// TIA Portal V19 export
FUNCTION "STOP PRODUCTION" : Void   // FC46, STL
TITLE = STOP PRODUCTION ASEPTIC TANK
{ S7_Optimized_Access := 'TRUE' }
NAME : SPROTNK
VERSION : 0.0
// Comment
// stored: AutoNumber false
BEGIN

NETWORK
TITLE = STOP PRODUCTION ASEPTIC TANK
// "M_PACK1", "M_PACK2", "M_PACK3", "M_PACK4" have been commented out to free up 
// outputs which were not wired, to be used for the Combi 512 Filler cip interface
      AN    "S0 STOP PRODUCTION TANK";
      R     "S1 STOP PRODUCTION TANK";
      R     "S2 STOP PRODUCTION TANK";
      BEC;
      A     "S1 STOP PRODUCTION TANK";
      JC    M001;
      R     "TANK STERILE";
      R     "MY0113";
      R     "MY0112";
      S     "MY0114";
      R     "MY0148";
      R     "IF_Device".V_09_30.IO.V._IO.IN.Activate;
      R     "IF_Device".V_09_31.IO.V._IO.IN.Activate;
      R     "TEST BARRIERS";
      R     "TEST FILLING PRESSURE";
//     R     "MM01.30"
      R     "START FILLING TANK";
      R     "STOP FILLING TANK";
      R     "MY0147";
      R     "M_AHV_READY";
//     R     "M_PACK1"
//     R     "M_PACK2"
//     R     "M_PACK3"
//     R     "M_PACK4"
      R     "DUMMY PROD. AT FILLING";
      R     "AGITATOR AUTOMATIC";
      R     "AGITATOR MANUEL";

//      A     "B01.66"
//      S     "A13-DRAIN THE TANK"
//      SET

      S     "S1 STOP PRODUCTION TANK";
      BEU;
M001: NOP   0;

NETWORK
TITLE = 
// Comment
      A     "S2 STOP PRODUCTION TANK";
      JC    c001;
//      A     "B01.66"
//      S     "A13-DRAIN THE TANK"
//      BEC
      S     "LEDAssignment".K4_FLASH;  //"FLASH_K4_CIP_LYE"
      R     "LEDAssignment".K4_LIGHT;  //"LIGHT_K4_CIP_LYE"
      S     "LEDAssignment".K5_FLASH;  //"FLASH_K5_CIP_LYE_ACID"
      R     "LEDAssignment".K5_LIGHT;  //"LIGHT_K5_CIP_LYE_ACID"
      R     "LEDAssignment".K7_FLASH;  //"FLASH_K7_STOP"
      R     "LEDAssignment".K7_LIGHT;  //"LIGHT_K7_STOP"
      S     "S2 STOP PRODUCTION TANK";
      BEU;
c001: NOP   0;
END_FUNCTION
